// TIA Portal project "Profinet_Test" (V19)

(* hardware
DEVICE "S7-1500/ET200MP station_1"  S7-1500 station
   slot 0: "Rail_0"  Rack  6ES7 590-1***0-0AA0
   slot 1: "PLC_1"  CPU 1516-3 PN/DP  6ES7 516-3AN01-0AB0  V2.9
      slot 3: "CPU display_1"  6ES7591-1BA00-0AA0
      slot 32768: "PROFINET interface_1"  X1
         slot 32769: "Port_1"  X1 P1
         slot 32770: "Port_2"  X1 P2
      slot 33024: "PROFINET interface_2"  X2
         slot 33025: "Port_1"  X2 P1
      slot 33280: "DP interface_1"  X3
      slot 34817: "Virtual CP interface port_1"  Virtual CP interface port  Virtual CP interface port
DEVICE "PROFINET Driver_1"  PROFINET Driver
   slot 0: "PC station"  PROFINET Driver Rack V2.2  6ES7 195-3***0-0YA0
   slot 1: "PROFINET Driver"  PROFINET Driver  6ES7 195-3AA00-0YA0  V2.2
      slot 32768: "PROFINET interface"  PN Driver Linux Native Submodule Interface  Linux Native  V2.2
         slot 1: "Port"  PN Driver Linux Native Port  V2.2
*)

// ===== PLC "PLC_1"  CPU 1516-3 PN/DP =====

VAR_GLOBAL   // PLC tag table "Default tag table"
   "iProfinetOutput" AT %QW0 : Int;
END_VAR

DATA_BLOCK "Data"   // DB1
{ S7_Optimized_Access := 'TRUE' }
VERSION : 0.1
   VAR
      iProfinetTest : Int;
   END_VAR
BEGIN
END_DATA_BLOCK

ORGANIZATION_BLOCK "Main"   // OB1, LAD, ProgramCycle
TITLE = "Main Program Sweep (Cycle)"
{ S7_Optimized_Access := 'TRUE' }
VERSION : 0.1
   VAR_INPUT
      Initial_Call : Bool;   // Initial call of this OB
      Remanence : Bool;   // =True, if remanent data are available
   END_VAR
BEGIN

REGION Network 1
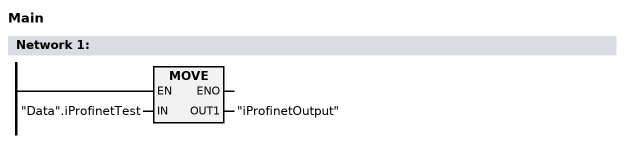
   RUNG wire#powerrail
      Move(in := "Data".iProfinetTest, out1 => "iProfinetOutput")
   END_RUNG
   // the same network as SCL:
   "iProfinetOutput" := "Data".iProfinetTest;
END_REGION
END_ORGANIZATION_BLOCK